SUBAPPLICATION Reset (* 1 Button, 1 Softkey *)
  (* Standard: 61499-2 *)
  (* Version 1.0, 2023-02-17, Franz *)
  PACKAGE FBs::Counter::subs::Buttons;
  IMPORT isobus::UT::Q::const::IDs::ID_NULL;
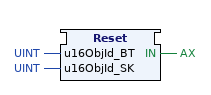
  VAR_INPUT
    u16ObjId_BT : UINT := ID_NULL; (* Object ID Button *)
    u16ObjId_SK : UINT := ID_NULL; (* Object ID SoftKey *)
  END_VAR
  PLUGS
    IN : adapter::types::unidirectional::AX;
  END_PLUGS
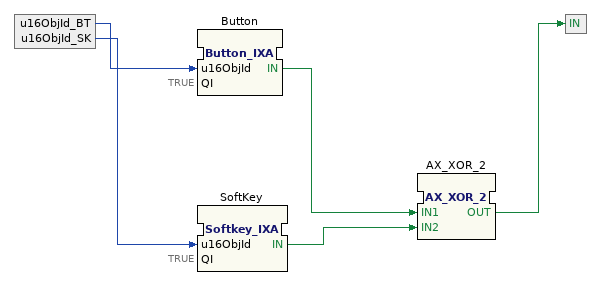
  FBS
    Button : isobus::UT::io::Button::Button_IXA(QI := TRUE);
    SoftKey : isobus::UT::io::Softkey::Softkey_IXA(QI := TRUE);
    AX_XOR_2 : adapter::booleanOperators::AX_XOR_2;
  END_FBS
  DATA_CONNECTIONS
    u16ObjId_BT TO Button.u16ObjId;
    u16ObjId_SK TO SoftKey.u16ObjId;
  END_CONNECTIONS
  ADAPTER_CONNECTIONS
    Button.IN TO AX_XOR_2.IN1;
    SoftKey.IN TO AX_XOR_2.IN2;
    AX_XOR_2.OUT TO IN;
  END_CONNECTIONS
END_SUBAPPLICATION
